FUNCTION_BLOCK FB_EventLoggerCore EXTENDS TcLogCore
VAR_INPUT
END_VAR
VAR_OUTPUT
END_VAR
VAR
END_VAR

END_FUNCTION_BLOCK

(* stored: Version 1.1.0.1, ProductVersion 3.1.4024.12
   POU FB_EventLoggerCore: Id {a3461c24-8d97-428e-b3cb-0fe3d91d5f29}, SpecialFunc None *)
